// LS Electric XG5000 project: 동남95
// PLC NewPLC
// module base 0 slot 0: 입출력 모듈:XBC-DN/DP14E (DC 24V 입력 8점, 트랜지스터 출력 6점)

PROGRAM NewProgram (task: 스캔 프로그램)

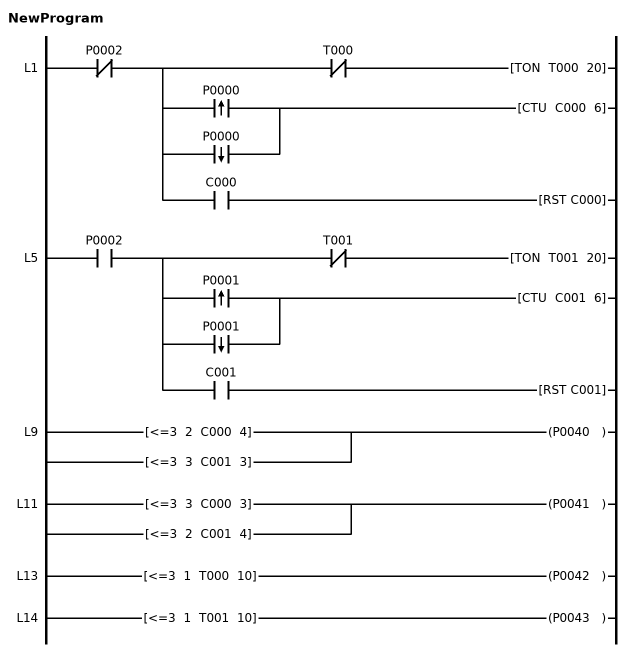
; L1
LOAD NOT  P0002
MPUSH
AND NOT   T000
TON       T000 20
MLOAD
LOADP     P0000
ORN       P0000
AND LOAD
CTU       C000 6
MPOP
AND       C000
RST       C000
; L5
LOAD      P0002
MPUSH
AND NOT   T001
TON       T001 20
MLOAD
LOADP     P0001
ORN       P0001
AND LOAD
CTU       C001 6
MPOP
AND       C001
RST       C001
; L9
LOAD<=3   2 C000 4
OR<=3     3 C001 3
OUT       P0040
; L11
LOAD<=3   3 C000 3
OR<=3     2 C001 4
OUT       P0041
; L13
LOAD<=3   1 T000 10
OUT       P0042
; L14
LOAD<=3   1 T001 10
OUT       P0043